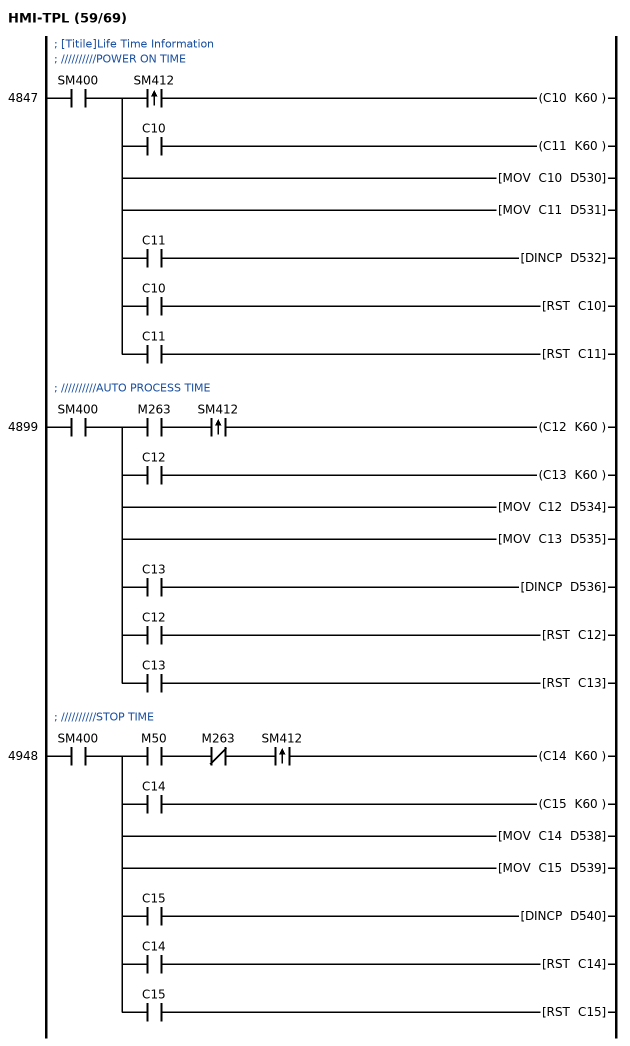
[picture p456: ladder of HMI-TPL, rungs at steps 4847 to 4948]
; [Titile]Life Time Information
; //////////POWER ON TIME
4847  LD      SM400
      MPS
      ANDP    SM412
      OUT     C10 K60
      MRD
      AND     C10
      OUT     C11 K60
      MPP
      MOV     C10 D530
      MOV     C11 D531
      MPS
      AND     C11
      DINCP   D532
      MRD
      AND     C10
      RST     C10
      MPP
      AND     C11
      RST     C11
; //////////AUTO PROCESS TIME
4899  LD      SM400
      MPS
      AND     M263
      ANDP    SM412
      OUT     C12 K60
      MRD
      AND     C12
      OUT     C13 K60
      MPP
      MOV     C12 D534
      MOV     C13 D535
      MPS
      AND     C13
      DINCP   D536
      MRD
      AND     C12
      RST     C12
      MPP
      AND     C13
      RST     C13
; //////////STOP TIME
4948  LD      SM400
      MPS
      AND     M50
      ANI     M263
      ANDP    SM412
      OUT     C14 K60
      MRD
      AND     C14
      OUT     C15 K60
      MPP
      MOV     C14 D538
      MOV     C15 D539
      MPS
      AND     C15
      DINCP   D540
      MRD
      AND     C14
      RST     C14
      MPP
      AND     C15
      RST     C15
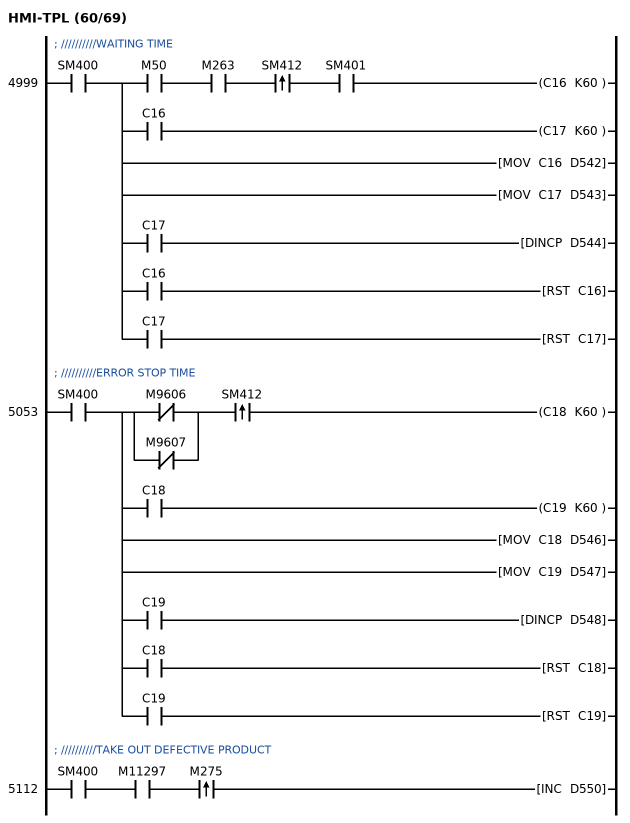
; //////////WAITING TIME
4999  LD      SM400
      MPS
      AND     M50
      AND     M263
      ANDP    SM412
      AND     SM401
      OUT     C16 K60
      MRD
      AND     C16
      OUT     C17 K60
      MPP
      MOV     C16 D542
      MOV     C17 D543
      MPS
      AND     C17
      DINCP   D544
      MRD
      AND     C16
      RST     C16
      MPP
      AND     C17
      RST     C17
; //////////ERROR STOP TIME
5053  LD      SM400
      MPS
      LDI     M9606
      ORI     M9607
      ANB
      ANDP    SM412
      OUT     C18 K60
      MRD
      AND     C18
      OUT     C19 K60
      MPP
      MOV     C18 D546
      MOV     C19 D547
      MPS
      AND     C19
      DINCP   D548
      MRD
      AND     C18
      RST     C18
      MPP
      AND     C19
      RST     C19
; //////////TAKE OUT DEFECTIVE PRODUCT
5112  LD      SM400
      AND     M11297
      ANDP    M275
      INC     D550
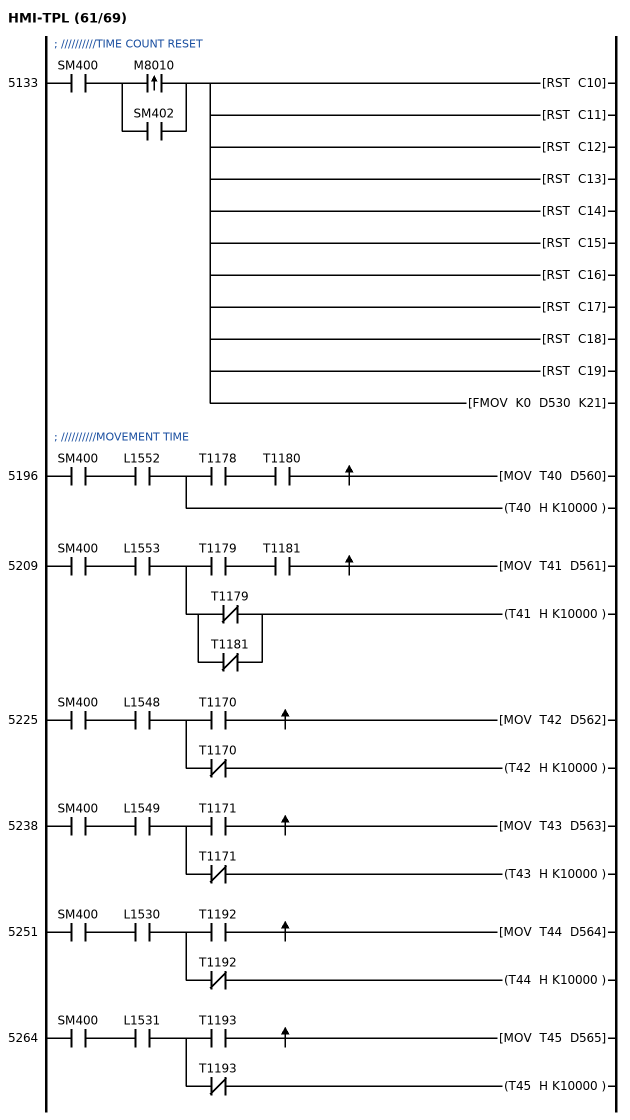
; //////////TIME COUNT RESET
5133  LD      SM400
      LDP     M8010
      OR      SM402
      ANB
      RST     C10
      RST     C11
      RST     C12
      RST     C13
      RST     C14
      RST     C15
      RST     C16
      RST     C17
      RST     C18
      RST     C19
      FMOV    K0 D530 K21
; //////////MOVEMENT TIME
5196  LD      SM400
      AND     L1552
      MPS
      AND     T1178
      AND     T1180
      MEP
      MOV     T40 D560
      MPP
      OUTH    T40 K10000
5209  LD      SM400
      AND     L1553
      MPS
      AND     T1179
      AND     T1181
      MEP
      MOV     T41 D561
      MPP
      LDI     T1179
      ORI     T1181
      ANB
      OUTH    T41 K10000
5225  LD      SM400
      AND     L1548
      MPS
      AND     T1170
      MEP
      MOV     T42 D562
      MPP
      ANI     T1170
      OUTH    T42 K10000
5238  LD      SM400
      AND     L1549
      MPS
      AND     T1171
      MEP
      MOV     T43 D563
      MPP
      ANI     T1171
      OUTH    T43 K10000
5251  LD      SM400
      AND     L1530
      MPS
      AND     T1192
      MEP
      MOV     T44 D564
      MPP
      ANI     T1192
      OUTH    T44 K10000
5264  LD      SM400
      AND     L1531
      MPS
      AND     T1193
      MEP
      MOV     T45 D565
      MPP
      ANI     T1193
      OUTH    T45 K10000
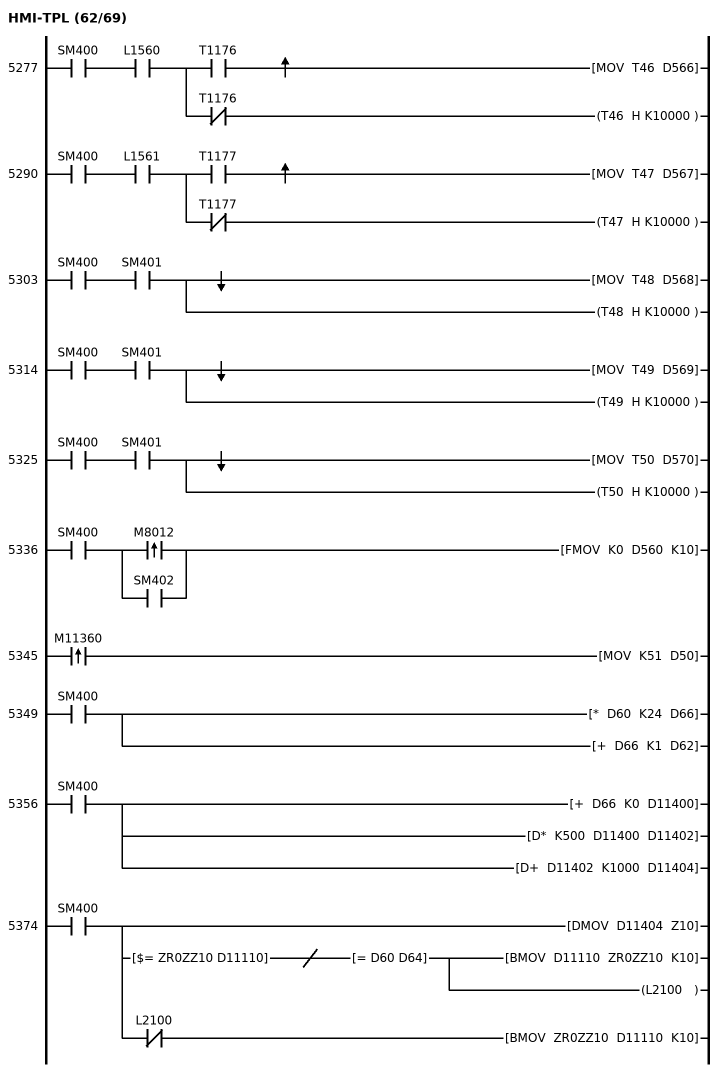
5277  LD      SM400
      AND     L1560
      MPS
      AND     T1176
      MEP
      MOV     T46 D566
      MPP
      ANI     T1176
      OUTH    T46 K10000
5290  LD      SM400
      AND     L1561
      MPS
      AND     T1177
      MEP
      MOV     T47 D567
      MPP
      ANI     T1177
      OUTH    T47 K10000
5303  LD      SM400
      AND     SM401
      MPS
      MEF
      MOV     T48 D568
      MPP
      OUTH    T48 K10000
5314  LD      SM400
      AND     SM401
      MPS
      MEF
      MOV     T49 D569
      MPP
      OUTH    T49 K10000
5325  LD      SM400
      AND     SM401
      MPS
      MEF
      MOV     T50 D570
      MPP
      OUTH    T50 K10000
5336  LD      SM400
      LDP     M8012
      OR      SM402
      ANB
      FMOV    K0 D560 K10
5345  LDP     M11360
      MOV     K51 D50
5349  LD      SM400
      *       D60 K24 D66
      +       D66 K1 D62
5356  LD      SM400
      +       D66 K0 D11400
        [note] row No.1
      D*      K500 D11400 D11402
      D+      D11402 K1000 D11404
5374  LD      SM400
      DMOV    D11404 Z10
      MPS
      AND$=   ZR0ZZ10 D11110
      INV
      AND=    D60 D64
      BMOV    D11110 ZR0ZZ10 K10
      OUT     L2100
      MPP
      ANI     L2100
      BMOV    ZR0ZZ10 D11110 K10
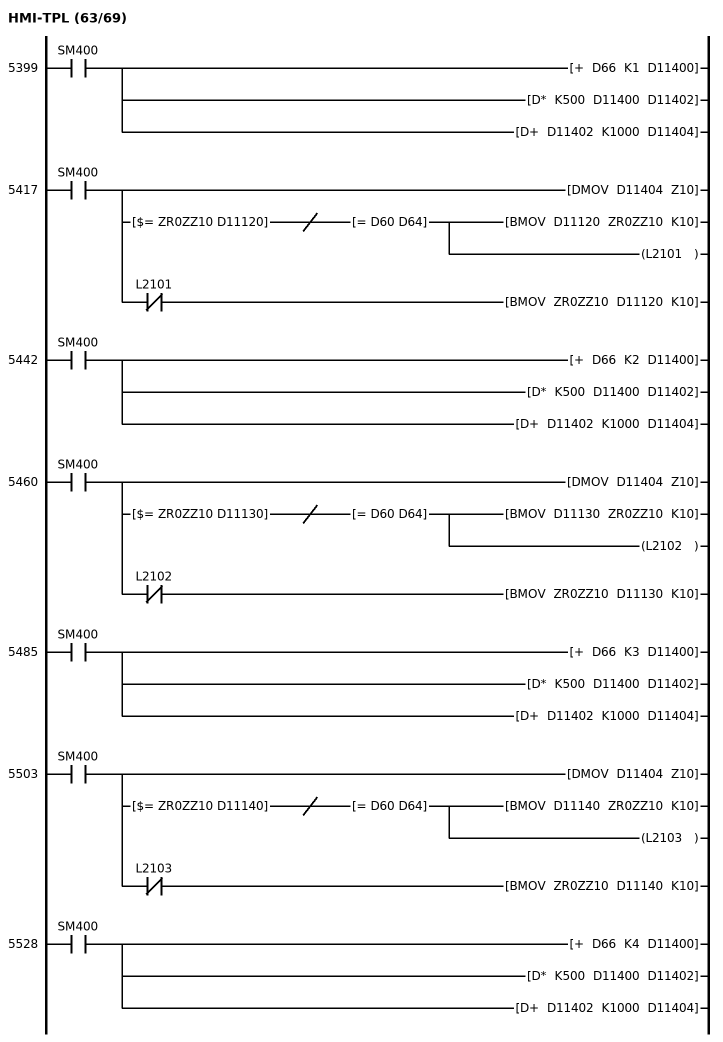
5399  LD      SM400
      +       D66 K1 D11400
        [note] row No.2
      D*      K500 D11400 D11402
      D+      D11402 K1000 D11404
5417  LD      SM400
      DMOV    D11404 Z10
      MPS
      AND$=   ZR0ZZ10 D11120
      INV
      AND=    D60 D64
      BMOV    D11120 ZR0ZZ10 K10
      OUT     L2101
      MPP
      ANI     L2101
      BMOV    ZR0ZZ10 D11120 K10
5442  LD      SM400
      +       D66 K2 D11400
        [note] row No.3
      D*      K500 D11400 D11402
      D+      D11402 K1000 D11404
5460  LD      SM400
      DMOV    D11404 Z10
      MPS
      AND$=   ZR0ZZ10 D11130
      INV
      AND=    D60 D64
      BMOV    D11130 ZR0ZZ10 K10
      OUT     L2102
      MPP
      ANI     L2102
      BMOV    ZR0ZZ10 D11130 K10
5485  LD      SM400
      +       D66 K3 D11400
        [note] row No.4
      D*      K500 D11400 D11402
      D+      D11402 K1000 D11404
5503  LD      SM400
      DMOV    D11404 Z10
      MPS
      AND$=   ZR0ZZ10 D11140
      INV
      AND=    D60 D64
      BMOV    D11140 ZR0ZZ10 K10
      OUT     L2103
      MPP
      ANI     L2103
      BMOV    ZR0ZZ10 D11140 K10
5528  LD      SM400
      +       D66 K4 D11400
        [note] row No.5
      D*      K500 D11400 D11402
      D+      D11402 K1000 D11404
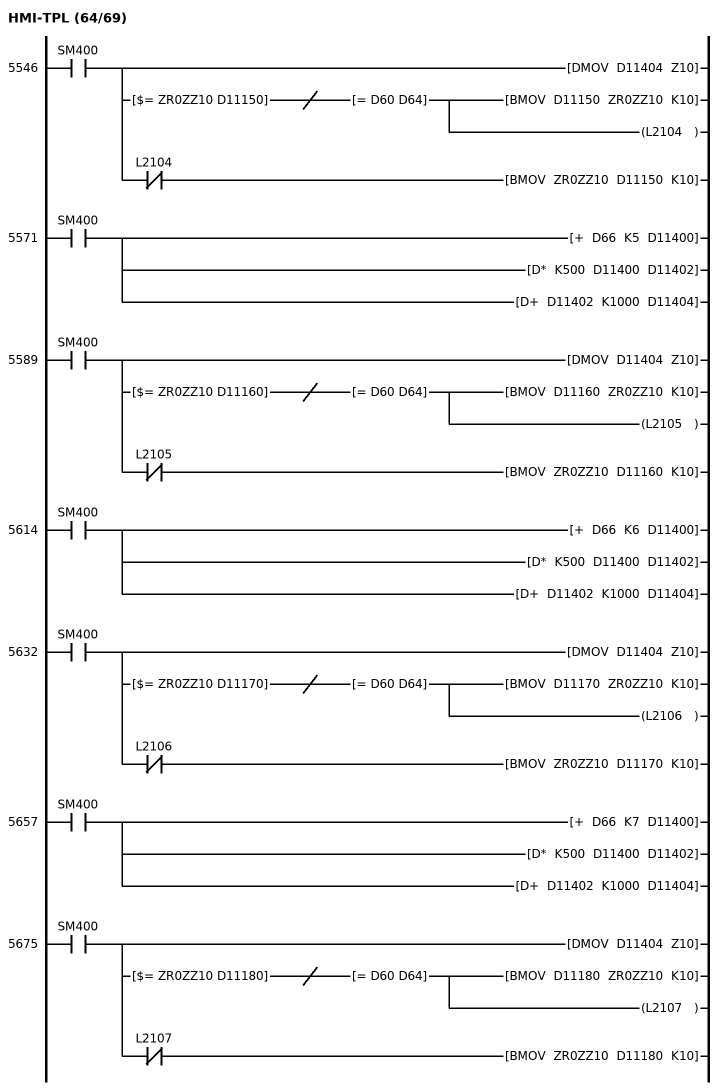
5546  LD      SM400
      DMOV    D11404 Z10
      MPS
      AND$=   ZR0ZZ10 D11150
      INV
      AND=    D60 D64
      BMOV    D11150 ZR0ZZ10 K10
      OUT     L2104
      MPP
      ANI     L2104
      BMOV    ZR0ZZ10 D11150 K10
5571  LD      SM400
      +       D66 K5 D11400
        [note] row No.6
      D*      K500 D11400 D11402
      D+      D11402 K1000 D11404
5589  LD      SM400
      DMOV    D11404 Z10
      MPS
      AND$=   ZR0ZZ10 D11160
      INV
      AND=    D60 D64
      BMOV    D11160 ZR0ZZ10 K10
      OUT     L2105
      MPP
      ANI     L2105
      BMOV    ZR0ZZ10 D11160 K10
5614  LD      SM400
      +       D66 K6 D11400
        [note] row No.7
      D*      K500 D11400 D11402
      D+      D11402 K1000 D11404
5632  LD      SM400
      DMOV    D11404 Z10
      MPS
      AND$=   ZR0ZZ10 D11170
      INV
      AND=    D60 D64
      BMOV    D11170 ZR0ZZ10 K10
      OUT     L2106
      MPP
      ANI     L2106
      BMOV    ZR0ZZ10 D11170 K10
5657  LD      SM400
      +       D66 K7 D11400
        [note] row No.8
      D*      K500 D11400 D11402
      D+      D11402 K1000 D11404
5675  LD      SM400
      DMOV    D11404 Z10
      MPS
      AND$=   ZR0ZZ10 D11180
      INV
      AND=    D60 D64
      BMOV    D11180 ZR0ZZ10 K10
      OUT     L2107
      MPP
      ANI     L2107
      BMOV    ZR0ZZ10 D11180 K10
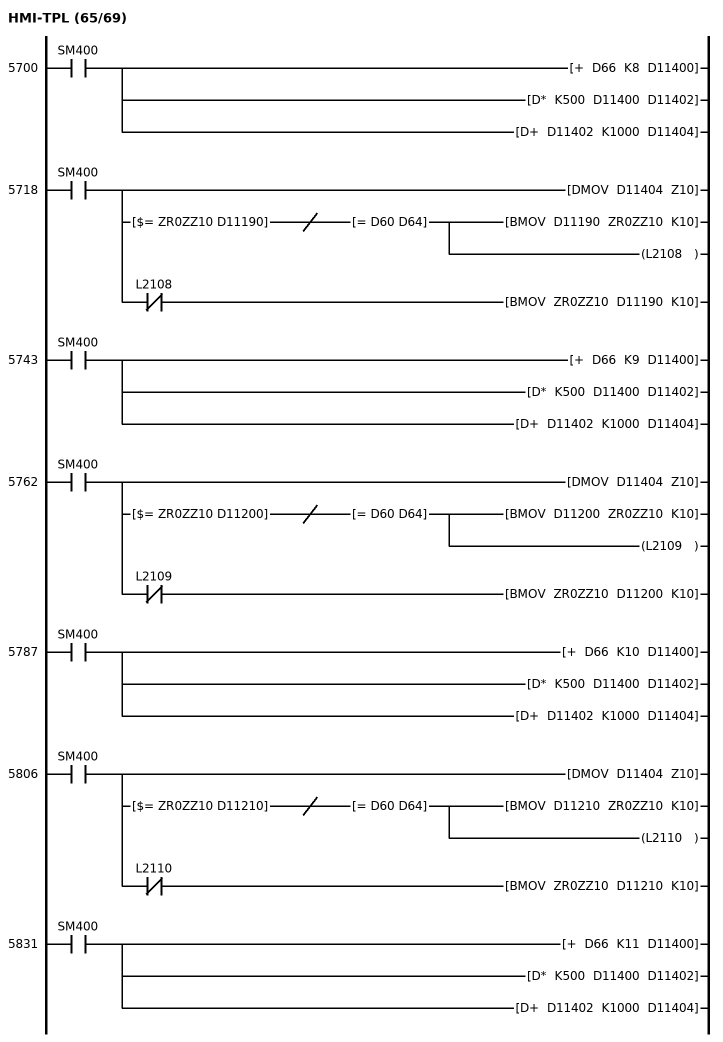
5700  LD      SM400
      +       D66 K8 D11400
        [note] row No.9
      D*      K500 D11400 D11402
      D+      D11402 K1000 D11404
5718  LD      SM400
      DMOV    D11404 Z10
      MPS
      AND$=   ZR0ZZ10 D11190
      INV
      AND=    D60 D64
      BMOV    D11190 ZR0ZZ10 K10
      OUT     L2108
      MPP
      ANI     L2108
      BMOV    ZR0ZZ10 D11190 K10
5743  LD      SM400
      +       D66 K9 D11400
        [note] row No.10
      D*      K500 D11400 D11402
      D+      D11402 K1000 D11404
5762  LD      SM400
      DMOV    D11404 Z10
      MPS
      AND$=   ZR0ZZ10 D11200
      INV
      AND=    D60 D64
      BMOV    D11200 ZR0ZZ10 K10
      OUT     L2109
      MPP
      ANI     L2109
      BMOV    ZR0ZZ10 D11200 K10
5787  LD      SM400
      +       D66 K10 D11400
        [note] row No.11
      D*      K500 D11400 D11402
      D+      D11402 K1000 D11404
5806  LD      SM400
      DMOV    D11404 Z10
      MPS
      AND$=   ZR0ZZ10 D11210
      INV
      AND=    D60 D64
      BMOV    D11210 ZR0ZZ10 K10
      OUT     L2110
      MPP
      ANI     L2110
      BMOV    ZR0ZZ10 D11210 K10
5831  LD      SM400
      +       D66 K11 D11400
        [note] row No.12
      D*      K500 D11400 D11402
      D+      D11402 K1000 D11404
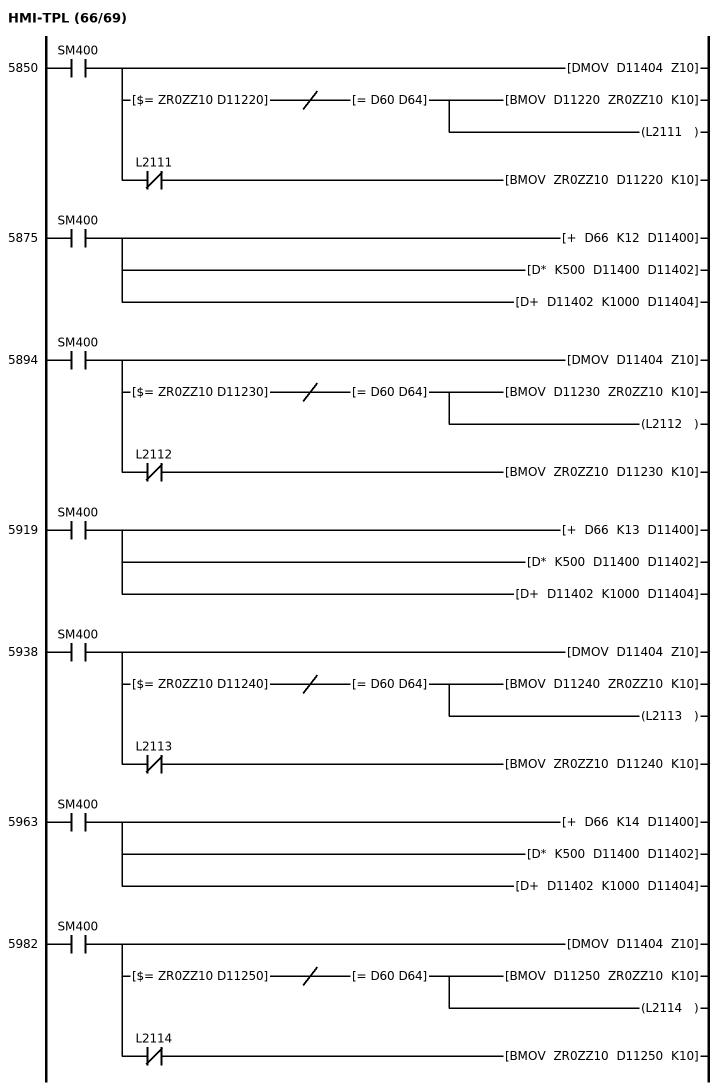
5850  LD      SM400
      DMOV    D11404 Z10
      MPS
      AND$=   ZR0ZZ10 D11220
      INV
      AND=    D60 D64
      BMOV    D11220 ZR0ZZ10 K10
      OUT     L2111
      MPP
      ANI     L2111
      BMOV    ZR0ZZ10 D11220 K10
5875  LD      SM400
      +       D66 K12 D11400
        [note] row No.13
      D*      K500 D11400 D11402
      D+      D11402 K1000 D11404
5894  LD      SM400
      DMOV    D11404 Z10
      MPS
      AND$=   ZR0ZZ10 D11230
      INV
      AND=    D60 D64
      BMOV    D11230 ZR0ZZ10 K10
      OUT     L2112
      MPP
      ANI     L2112
      BMOV    ZR0ZZ10 D11230 K10
5919  LD      SM400
      +       D66 K13 D11400
        [note] row No.14
      D*      K500 D11400 D11402
      D+      D11402 K1000 D11404
5938  LD      SM400
      DMOV    D11404 Z10
      MPS
      AND$=   ZR0ZZ10 D11240
      INV
      AND=    D60 D64
      BMOV    D11240 ZR0ZZ10 K10
      OUT     L2113
      MPP
      ANI     L2113
      BMOV    ZR0ZZ10 D11240 K10
5963  LD      SM400
      +       D66 K14 D11400
        [note] row No.15
      D*      K500 D11400 D11402
      D+      D11402 K1000 D11404
5982  LD      SM400
      DMOV    D11404 Z10
      MPS
      AND$=   ZR0ZZ10 D11250
      INV
      AND=    D60 D64
      BMOV    D11250 ZR0ZZ10 K10
      OUT     L2114
      MPP
      ANI     L2114
      BMOV    ZR0ZZ10 D11250 K10
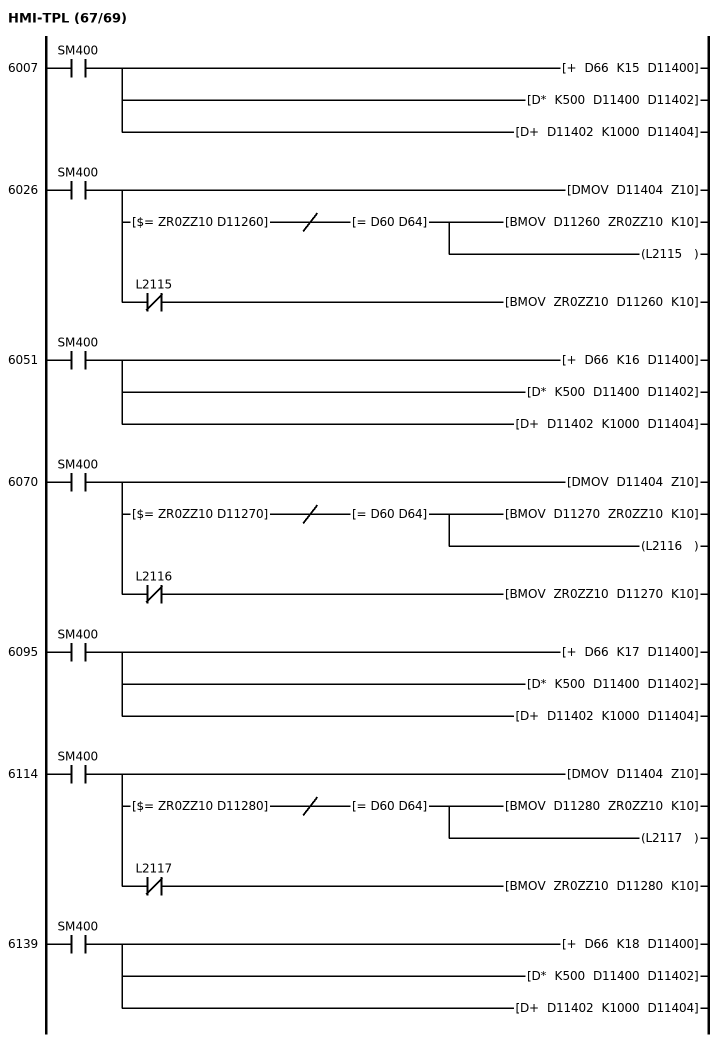
6007  LD      SM400
      +       D66 K15 D11400
        [note] row No.16
      D*      K500 D11400 D11402
      D+      D11402 K1000 D11404
6026  LD      SM400
      DMOV    D11404 Z10
      MPS
      AND$=   ZR0ZZ10 D11260
      INV
      AND=    D60 D64
      BMOV    D11260 ZR0ZZ10 K10
      OUT     L2115
      MPP
      ANI     L2115
      BMOV    ZR0ZZ10 D11260 K10
6051  LD      SM400
      +       D66 K16 D11400
        [note] row No.17
      D*      K500 D11400 D11402
      D+      D11402 K1000 D11404
6070  LD      SM400
      DMOV    D11404 Z10
      MPS
      AND$=   ZR0ZZ10 D11270
      INV
      AND=    D60 D64
      BMOV    D11270 ZR0ZZ10 K10
      OUT     L2116
      MPP
      ANI     L2116
      BMOV    ZR0ZZ10 D11270 K10
6095  LD      SM400
      +       D66 K17 D11400
        [note] row No.18
      D*      K500 D11400 D11402
      D+      D11402 K1000 D11404
6114  LD      SM400
      DMOV    D11404 Z10
      MPS
      AND$=   ZR0ZZ10 D11280
      INV
      AND=    D60 D64
      BMOV    D11280 ZR0ZZ10 K10
      OUT     L2117
      MPP
      ANI     L2117
      BMOV    ZR0ZZ10 D11280 K10
6139  LD      SM400
      +       D66 K18 D11400
        [note] row No.19
      D*      K500 D11400 D11402
      D+      D11402 K1000 D11404
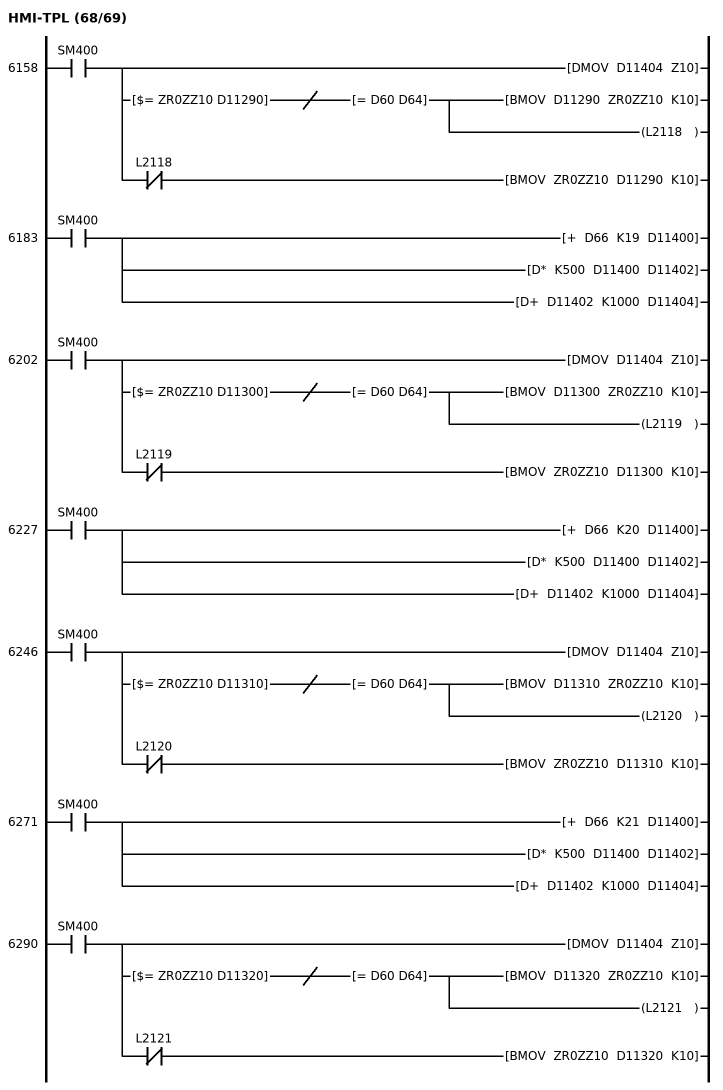
6158  LD      SM400
      DMOV    D11404 Z10
      MPS
      AND$=   ZR0ZZ10 D11290
      INV
      AND=    D60 D64
      BMOV    D11290 ZR0ZZ10 K10
      OUT     L2118
      MPP
      ANI     L2118
      BMOV    ZR0ZZ10 D11290 K10
6183  LD      SM400
      +       D66 K19 D11400
        [note] row No.20
      D*      K500 D11400 D11402
      D+      D11402 K1000 D11404
6202  LD      SM400
      DMOV    D11404 Z10
      MPS
      AND$=   ZR0ZZ10 D11300
      INV
      AND=    D60 D64
      BMOV    D11300 ZR0ZZ10 K10
      OUT     L2119
      MPP
      ANI     L2119
      BMOV    ZR0ZZ10 D11300 K10
6227  LD      SM400
      +       D66 K20 D11400
        [note] row No.21
      D*      K500 D11400 D11402
      D+      D11402 K1000 D11404
6246  LD      SM400
      DMOV    D11404 Z10
      MPS
      AND$=   ZR0ZZ10 D11310
      INV
      AND=    D60 D64
      BMOV    D11310 ZR0ZZ10 K10
      OUT     L2120
      MPP
      ANI     L2120
      BMOV    ZR0ZZ10 D11310 K10
6271  LD      SM400
      +       D66 K21 D11400
        [note] row No.22
      D*      K500 D11400 D11402
      D+      D11402 K1000 D11404
6290  LD      SM400
      DMOV    D11404 Z10
      MPS
      AND$=   ZR0ZZ10 D11320
      INV
      AND=    D60 D64
      BMOV    D11320 ZR0ZZ10 K10
      OUT     L2121
      MPP
      ANI     L2121
      BMOV    ZR0ZZ10 D11320 K10
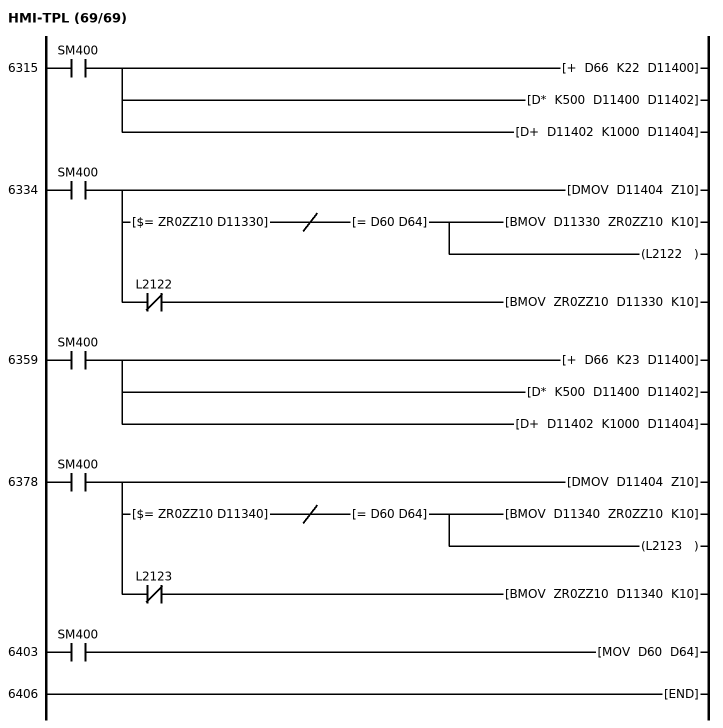
6315  LD      SM400
      +       D66 K22 D11400
        [note] row No.23
      D*      K500 D11400 D11402
      D+      D11402 K1000 D11404
6334  LD      SM400
      DMOV    D11404 Z10
      MPS
      AND$=   ZR0ZZ10 D11330
      INV
      AND=    D60 D64
      BMOV    D11330 ZR0ZZ10 K10
      OUT     L2122
      MPP
      ANI     L2122
      BMOV    ZR0ZZ10 D11330 K10
6359  LD      SM400
      +       D66 K23 D11400
        [note] row No.24
      D*      K500 D11400 D11402
      D+      D11402 K1000 D11404
6378  LD      SM400
      DMOV    D11404 Z10
      MPS
      AND$=   ZR0ZZ10 D11340
      INV
      AND=    D60 D64
      BMOV    D11340 ZR0ZZ10 K10
      OUT     L2123
      MPP
      ANI     L2123
      BMOV    ZR0ZZ10 D11340 K10
6403  LD      SM400
      MOV     D60 D64
6406  END
END_PROGRAM
